// TIA Portal V18 export
// export: Created 2025-12-01T12:38:02.9386683Z, ExportSetting None, DisplayName Totally Integrated Automation Portal, DisplayVersion V18 Update 5, DisplayName TIA Portal Openness, DisplayVersion V18 Update 5, DisplayName TIA Portal Teamcenter Gateway, DisplayVersion V18, DisplayName TIA Portal Version Control Interface, DisplayVersion V18, DisplayName STEP 7 Professional, DisplayVersion V18 Update 5, DisplayName STEP 7 Safety, DisplayVersion V18, DisplayName WinCC Professional, DisplayVersion V18 Update 5
FUNCTION_BLOCK "FB_Analog"   // FB4090, LAD
{ S7_Optimized_Access := 'TRUE' }
// stored: AutoNumber false, MemoryReserve 100, SetENOAutomatically false
   VAR_INPUT
      iSysInface : "RCS_SysComInterface_V1";
      "iunit in" : UInt;   // 0:mA(电流);1:V(电压)
      "iunit out" : UInt;   // 0:mm(毫米);1:N(牛顿);2.KN(千牛顿);3.bar(帕);4:kPa;5:mbar;6:bar;7:m/s;8:°
      "iHardware input" : Word;   // 硬件输入
      iRangeDown : Real;
      iRangeUp : Real;
   END_VAR
   VAR_IN_OUT
      io_Dev : "ST_GeneralAnalog";
   END_VAR
   VAR_TEMP
      TmpMidReal0 : Real;
   END_VAR
BEGIN

REGION Network 1: 启动条件 / Starting condition
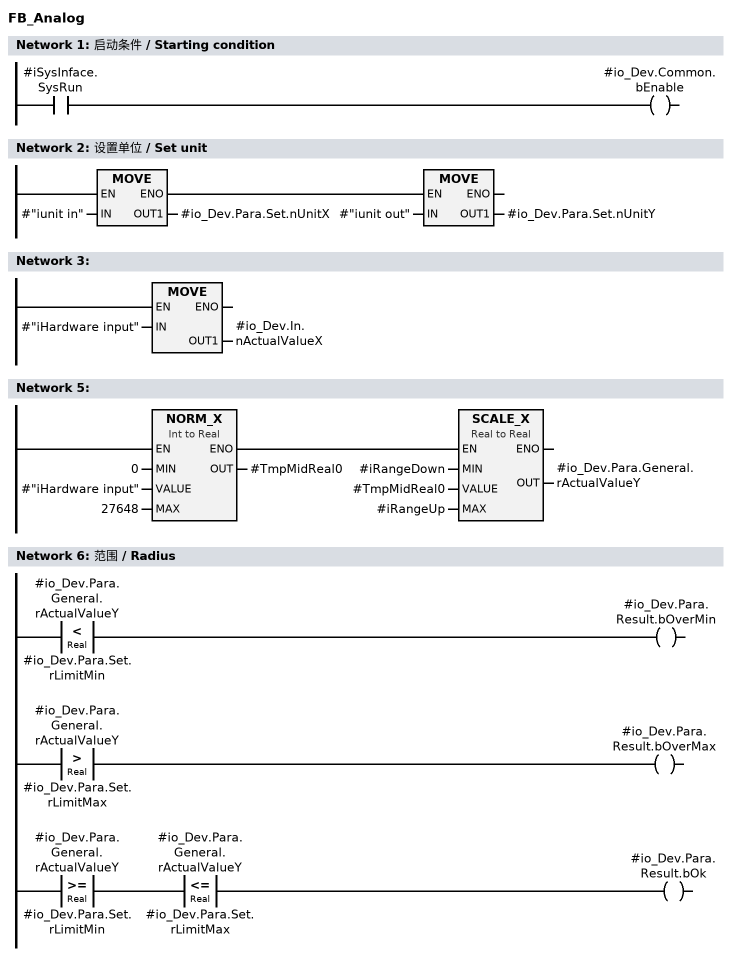
   RUNG wire#powerrail
      Contact( #iSysInface.SysRun )
      Coil( #io_Dev.Common.bEnable )
   END_RUNG
   // the same network as SCL:
   #io_Dev.Common.bEnable := #iSysInface.SysRun;
END_REGION

REGION Network 2: 设置单位 / Set unit
   RUNG wire#powerrail
      Move(in := #"iunit in", out1 => #io_Dev.Para.Set.nUnitX)
      Move(in := #"iunit out", out1 => #io_Dev.Para.Set.nUnitY)
   END_RUNG
   // the same network as SCL:
   #io_Dev.Para.Set.nUnitX := #"iunit in";
   #io_Dev.Para.Set.nUnitY := #"iunit out";
END_REGION

REGION Network 3
   RUNG wire#powerrail
      Move(in := #"iHardware input", out1 => #io_Dev.In.nActualValueX)
   END_RUNG
   // the same network as SCL:
   #io_Dev.In.nActualValueX := #"iHardware input";
END_REGION

REGION Network 5
   RUNG wire#powerrail
      { S7_Templates := "[SrcType := Int, DestType := Real]" } Normalize(min := 0, value := #"iHardware input", max := 27648, out => #TmpMidReal0)
      { S7_Templates := "[SrcType := Real, DestType := Real]" } Scale(min := #iRangeDown, value := #TmpMidReal0, max := #iRangeUp, out => #io_Dev.Para.General.rActualValueY)
   END_RUNG
   // the same network as SCL:
   #TmpMidReal0 := NORM_X(MIN := 0, VALUE := #"iHardware input", MAX := 27648);
   #io_Dev.Para.General.rActualValueY := SCALE_X(MIN := #iRangeDown, VALUE := #TmpMidReal0, MAX := #iRangeUp);
END_REGION

REGION Network 6: 范围 / Radius
   RUNG wire#powerrail
      { S7_Templates := "SrcType := Real" } LT_Contact(in1 := #io_Dev.Para.General.rActualValueY, in2 := #io_Dev.Para.Set.rLimitMin)
      Coil( #io_Dev.Para.Result.bOverMin )
   END_RUNG
   RUNG wire#powerrail
      { S7_Templates := "SrcType := Real" } GT_Contact(in1 := #io_Dev.Para.General.rActualValueY, in2 := #io_Dev.Para.Set.rLimitMax)
      Coil( #io_Dev.Para.Result.bOverMax )
   END_RUNG
   RUNG wire#powerrail
      { S7_Templates := "SrcType := Real" } GE_Contact(in1 := #io_Dev.Para.General.rActualValueY, in2 := #io_Dev.Para.Set.rLimitMin)
      { S7_Templates := "SrcType := Real" } LE_Contact(in1 := #io_Dev.Para.General.rActualValueY, in2 := #io_Dev.Para.Set.rLimitMax)
      Coil( #io_Dev.Para.Result.bOk )
   END_RUNG
   // the same network as SCL:
   #io_Dev.Para.Result.bOverMin := #io_Dev.Para.General.rActualValueY < #io_Dev.Para.Set.rLimitMin;
   #io_Dev.Para.Result.bOverMax := #io_Dev.Para.General.rActualValueY > #io_Dev.Para.Set.rLimitMax;
   #io_Dev.Para.Result.bOk := (#io_Dev.Para.General.rActualValueY >= #io_Dev.Para.Set.rLimitMin) AND (#io_Dev.Para.General.rActualValueY <= #io_Dev.Para.Set.rLimitMax);
END_REGION
END_FUNCTION_BLOCK
